INTERFACE INTERNAL _I_Execute EXTENDS I_Debug, I_ValidateInterface;

METHOD INTERNAL _Exe
VAR_OUTPUT
	iNext: _I_Execute;
END_VAR
END_METHOD

METHOD INTERNAL GetNext : _I_Execute
END_METHOD

METHOD INTERNAL SetNext
VAR_INPUT
	iNext: _I_Execute;
END_VAR
END_METHOD

METHOD INTERNAL GetPrev : _I_Execute
END_METHOD

METHOD INTERNAL SetPrev
VAR_INPUT
	iPrev: _I_Execute;
END_VAR
END_METHOD

METHOD INTERNAL GetThread : I_Thread
END_METHOD

METHOD INTERNAL SetThread
VAR_INPUT
	iThread: I_Thread;
END_VAR
END_METHOD

END_INTERFACE

(* stored: Version 1.1.0.1
   Itf _I_Execute: Id {8b79cbd5-d7c4-4c85-85bb-38aa830221fc}
   Method _Exe: Id {8d48a61b-dcd6-4e45-8916-d669dffef6c5}
   Method GetNext: Id {5b543610-e1fa-4f2b-a8a0-54202ae4a9dc}
   Method SetNext: Id {ac7fcdda-3d58-45fe-b3c7-62ee13cdb491}
   Method GetPrev: Id {8ec9a1af-7511-4197-89bc-92c02af4d758}
   Method SetPrev: Id {56724861-3fee-415a-a57c-8f1a19c2647b}
   Method GetThread: Id {135e4469-81eb-4248-a642-31db2477d4be}
   Method SetThread: Id {76dab680-b561-44e5-a302-e9e92c47b7f6} *)
